{attribute 'reflection'}
FUNCTION_BLOCK PUBLIC FB_ELModuleDiag
VAR_INPUT
END_VAR
VAR_OUTPUT
	bError 	:	BOOL ; // Module is in error
	sErrorDiscription : STRING ; // module error discription 
END_VAR
VAR
END_VAR

END_FUNCTION_BLOCK

(* stored: Version 1.1.0.1, ProductVersion 3.1.4024.5
   POU FB_ELModuleDiag: Id {7c3b6cf0-4cbb-0cc9-1d0a-bf4eda696d1d}, SpecialFunc None *)
